PROGRAM main
  VAR
    COUNTER1 AT %QW0 : INT;
    STATUS_BIT AT %QX0.0 : BOOL;
    TICK : BOOL;
    CALISMA_BITTI : BOOL;
    T_1S : TON;
    C1 : CTU;
    T_DURUS : TON;
    T_CALISMA : TON;
    REJECT_COUNTER AT %QW1 : INT;
    URETIM_DARBE : BOOL;
    C1_DOLU : BOOL;
    PARCA_20 : BOOL;
    HATA_DOLU : BOOL;
    C_PARCA : CTU;
    C_HATA : CTU;
    URET : BOOL;
    CTU0 : CTU;
    CTU1 : CTU;
  END_VAR

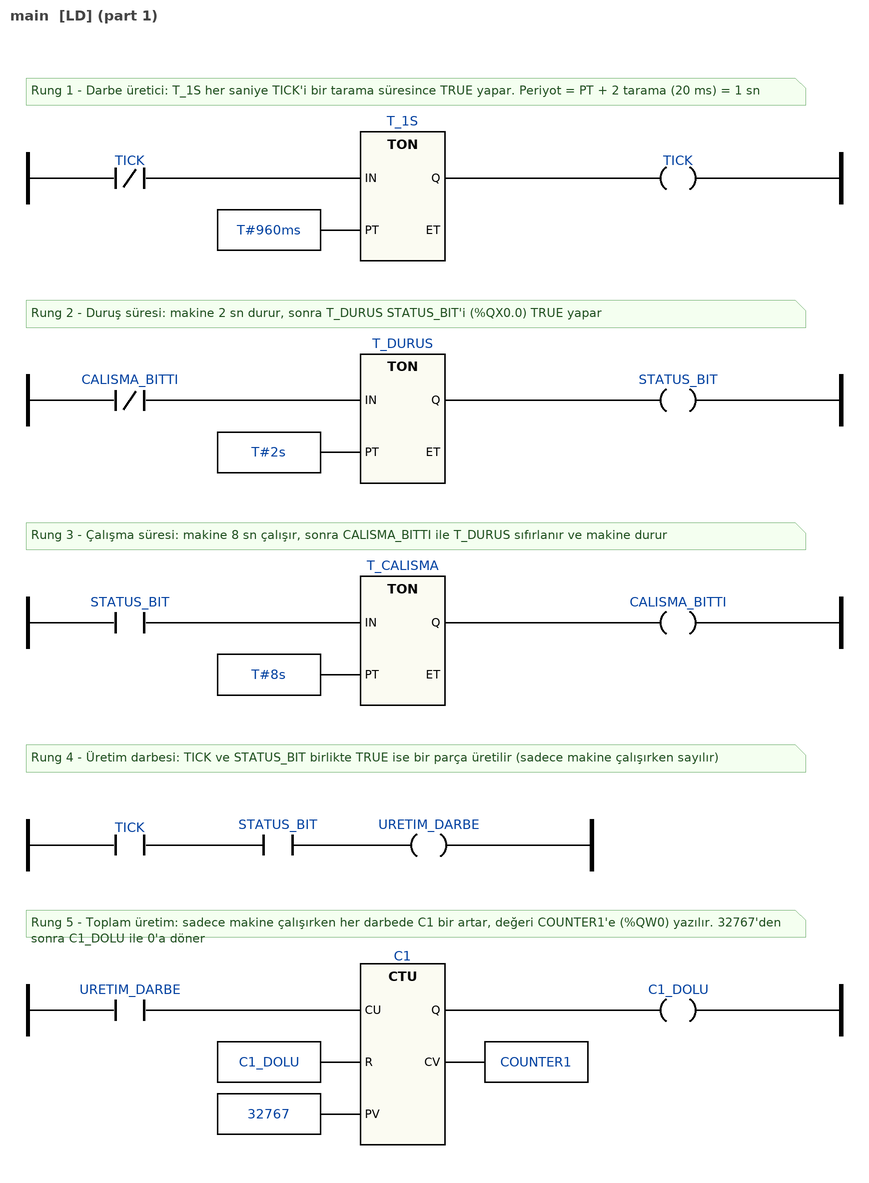
(* LD diagram, written out as Structured Text *)
(* Rung 1 - Darbe üretici: T_1S her saniye TICK'i bir tarama süresince TRUE yapar. Periyot = PT + 2 tarama (20 ms) = 1 sn *)
T_1S(IN := NOT TICK, PT := T#960ms);
TICK := T_1S.Q;
(* Rung 2 - Duruş süresi: makine 2 sn durur, sonra T_DURUS STATUS_BIT'i (%QX0.0) TRUE yapar *)
T_DURUS(IN := NOT CALISMA_BITTI, PT := T#2s);
STATUS_BIT := T_DURUS.Q;
(* Rung 3 - Çalışma süresi: makine 8 sn çalışır, sonra CALISMA_BITTI ile T_DURUS sıfırlanır ve makine durur *)
T_CALISMA(IN := STATUS_BIT, PT := T#8s);
CALISMA_BITTI := T_CALISMA.Q;
(* Rung 4 - Üretim darbesi: TICK ve STATUS_BIT birlikte TRUE ise bir parça üretilir (sadece makine çalışırken sayılır) *)
URETIM_DARBE := TICK AND STATUS_BIT;
(* Rung 5 - Toplam üretim: sadece makine çalışırken her darbede C1 bir artar, değeri COUNTER1'e (%QW0) yazılır. 32767'den sonra C1_DOLU ile 0'a döner *)
C1(CU := URETIM_DARBE, R := C1_DOLU, PV := 32767);
C1_DOLU := C1.Q;
COUNTER1 := C1.CV;
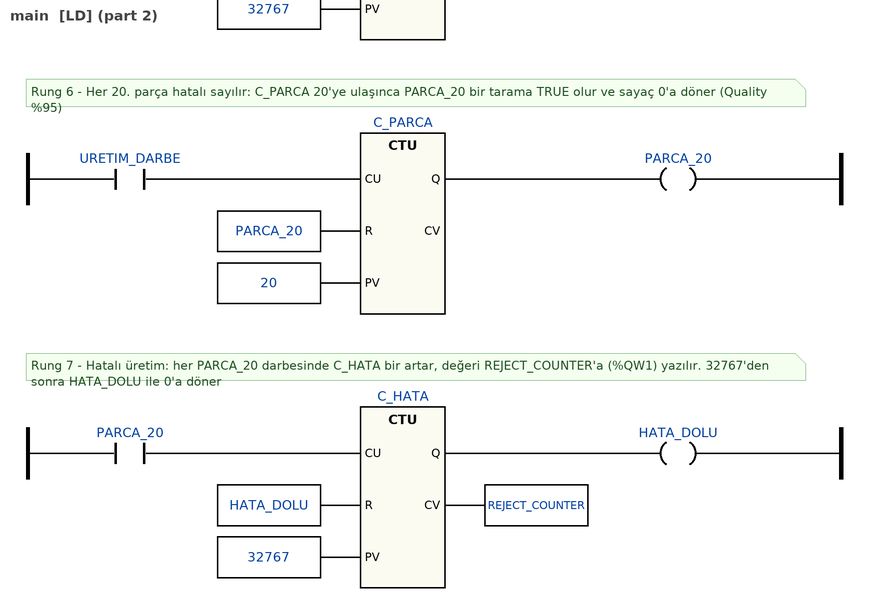
(* Rung 6 - Her 20. parça hatalı sayılır: C_PARCA 20'ye ulaşınca PARCA_20 bir tarama TRUE olur ve sayaç 0'a döner (Quality %95) *)
C_PARCA(CU := URETIM_DARBE, R := PARCA_20, PV := 20);
PARCA_20 := C_PARCA.Q;
(* Rung 7 - Hatalı üretim: her PARCA_20 darbesinde C_HATA bir artar, değeri REJECT_COUNTER'a (%QW1) yazılır. 32767'den sonra HATA_DOLU ile 0'a döner *)
C_HATA(CU := PARCA_20, R := HATA_DOLU, PV := 32767);
HATA_DOLU := C_HATA.Q;
REJECT_COUNTER := C_HATA.CV;
END_PROGRAM
